FUNCTION_BLOCK Btn_lock (* Basic Function Block Type *)
  (* Standard: 61499-2 *)
  (* Version 0.0, 7/27/2023, vv263, nxtControl GmBH, Template *)
  PACKAGE Main;
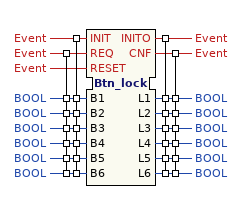
  EVENT_INPUT
    INIT WITH B1, B2, B3, B4, B5, B6; (* Initialization Request *)
    REQ WITH B1, B2, B3, B4, B5, B6; (* Normal Execution Request *)
    RESET;
  END_EVENT
  EVENT_OUTPUT
    INITO WITH L1, L2, L3, L4, L5, L6; (* Initialization Confirm *)
    CNF WITH L1, L2, L3, L4, L5, L6; (* Execution Confirmation *)
  END_EVENT
  VAR_INPUT
    B1 : BOOL; (* Input event qualifier *)
    B2 : BOOL;
    B3 : BOOL;
    B4 : BOOL;
    B5 : BOOL;
    B6 : BOOL;
  END_VAR
  VAR_OUTPUT
    L1 : BOOL; (* Output event qualifier *)
    L2 : BOOL;
    L3 : BOOL;
    L4 : BOOL;
    L5 : BOOL;
    L6 : BOOL;
  END_VAR
  VAR
    NumOn : INT;
    NumLitOn : INT;
  END_VAR
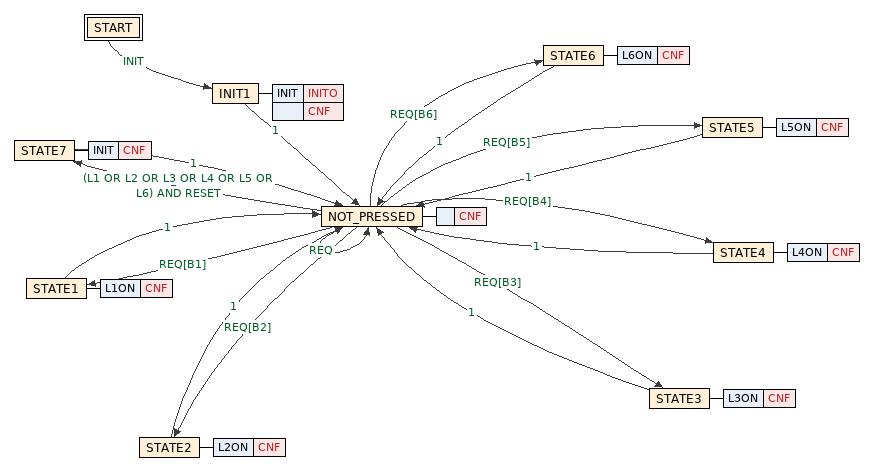
  EC_STATES
    START; (* Initial State *)
    NOT_PRESSED : -> CNF; (* Initialization *)
    STATE2 : L2ON -> CNF;
    STATE3 : L3ON -> CNF;
    STATE4 : L4ON -> CNF;
    STATE5 : L5ON -> CNF;
    STATE6 : L6ON -> CNF;
    INIT1 : INIT -> INITO, -> CNF;
    STATE1 : L1ON -> CNF;
    STATE7 : INIT -> CNF;
  END_STATES
  EC_TRANSITIONS
    START TO INIT1 := INIT;
    NOT_PRESSED TO STATE2 := REQ[B2];
    NOT_PRESSED TO STATE3 := REQ[B3];
    NOT_PRESSED TO STATE4 := REQ[B4];
    NOT_PRESSED TO STATE5 := REQ[B5];
    NOT_PRESSED TO STATE6 := REQ[B6];
    STATE2 TO NOT_PRESSED := 1;
    INIT1 TO NOT_PRESSED := 1;
    STATE1 TO NOT_PRESSED := 1;
    NOT_PRESSED TO STATE1 := REQ[B1];
    NOT_PRESSED TO STATE7 := (L1 OR L2 OR L3 OR L4 OR L5 OR L6) AND RESET;
    STATE7 TO NOT_PRESSED := 1;
    STATE3 TO NOT_PRESSED := 1;
    STATE4 TO NOT_PRESSED := 1;
    STATE5 TO NOT_PRESSED := 1;
    STATE6 TO NOT_PRESSED := 1;
    NOT_PRESSED TO NOT_PRESSED := REQ;
  END_TRANSITIONS
  ALGORITHM INIT IN ST: (* Initialization algorithm *)
L1:=FALSE;
L2:=FALSE;
L3:=FALSE;
L4:=FALSE;
L5:=FALSE;
L6:=FALSE;
  END_ALGORITHM
  ALGORITHM L1ON IN ST:
;
L1:=TRUE;
L2:=FALSE;
L3:=FALSE;
L4:=FALSE;
L5:=FALSE;
L6:=FALSE;
  END_ALGORITHM
  ALGORITHM L2ON IN ST:
;
L1:=FALSE;
L2:=TRUE;
L3:=FALSE;
L4:=FALSE;
L5:=FALSE;
L6:=FALSE;
  END_ALGORITHM
  ALGORITHM L3ON IN ST:
;
L1:=FALSE;
L2:=FALSE;
L3:=TRUE;
L4:=FALSE;
L5:=FALSE;
L6:=FALSE;
  END_ALGORITHM
  ALGORITHM L4ON IN ST:
;
L1:=FALSE;
L2:=FALSE;
L3:=FALSE;
L4:=TRUE;
L5:=FALSE;
L6:=FALSE;
  END_ALGORITHM
  ALGORITHM L5ON IN ST:
;
L1:=FALSE;
L2:=FALSE;
L3:=FALSE;
L4:=FALSE;
L5:=TRUE;
L6:=FALSE;
  END_ALGORITHM
  ALGORITHM L6ON IN ST:
;
L1:=FALSE;
L2:=FALSE;
L3:=FALSE;
L4:=FALSE;
L5:=FALSE;
L6:=TRUE;
  END_ALGORITHM
END_FUNCTION_BLOCK
